TYPE ST_ProductData :
STRUCT
	
	nSerial				: UDINT;
	bInitRun			: BOOL;
	nDestinationProcess	: UINT;
	nPriority			: UINT;
	

END_STRUCT
END_TYPE

(* stored: Version 1.1.0.1, ProductVersion 3.1.4024.5
   DUT ST_ProductData: Id {bdd20773-de6a-4c9e-8898-66bcede34983} *)
